FUNCTION_BLOCK ObserveSSC EXTENDS HardwareObservationBase
VAR_INPUT
END_VAR
VAR_OUTPUT
END_VAR
VAR
	m_ptrSSC: POINTER TO SmallSortingConveyor;
	m_ptrSSCWP1: POINTER TO xPPUProduct;
	m_ptrSSCWP2: POINTER TO xPPUProduct;
	
	m_rtWpAtRamp: R_TRIG;
END_VAR

METHOD FB_init : BOOL
VAR_INPUT
	bInitRetains : BOOL; // if TRUE, the retain variables are initialized (warm start / cold start)
	bInCopyCode : BOOL;  // if TRUE, the instance afterwards gets moved into the copy code (online change)
	
	i_ptrSSC: POINTER TO SmallSortingConveyor;
	i_ptrWP1: POINTER TO IProduct;
	i_ptrWP2: POINTER TO IProduct;
END_VAR
m_ptrSSC := i_ptrSSC;
IF NOT __QUERYPOINTER(i_ptrWP1^, m_ptrSSCWP1) THEN
	FB_init := FALSE;
END_IF
IF NOT __QUERYPOINTER(i_ptrWP2^, m_ptrSSCWP2) THEN
	FB_init := FALSE;
END_IF
END_METHOD

METHOD  ResetDefinition : BOOL
VAR_INPUT
END_VAR
;
END_METHOD

(* Update an instance of ProcessState with the part of the process that can be observed by this Hardware Interface. *)
METHOD UpdateProcessObservation : BOOL
VAR_IN_OUT
	io_processState: ProcessState;
END_VAR
m_rtWpAtRamp(CLK := m_ptrSSC^.WPAtRampEnd);

io_processState.UpdateState_Binary(EProcessVariables.SSC_WPAtStart, m_ptrSSC^.WPAtStart, TRUE);
io_processState.UpdateState_Binary(EProcessVariables.SSC_WPAtEnd, m_ptrSSC^.WPAtEnd, TRUE);
io_processState.UpdateState_Binary(EProcessVariables.SSC_WPLightAtMiddle, m_ptrSSC^.LightWPAtMid, TRUE);
io_processState.UpdateState_Binary(EProcessVariables.SSC_WPMetalAtMiddle, m_ptrSSC^.MetalWPAtMid, TRUE);
io_processState.UpdateState_Binary(EProcessVariables.SSC_WPAtRampEnd, m_ptrSSC^.WPAtRampEnd, TRUE);
io_processState.UpdateState_Binary(EProcessVariables.SSC_SwitchExtended, m_ptrSSC^.m_Switch.Extended, TRUE);
io_processState.UpdateState_Binary(EProcessVariables.SSC_SwitchRetracted, m_ptrSSC^.m_Switch.Retracted, TRUE);

IF m_rtWpAtRamp.Q THEN
	io_processState.UpdateState_NumericIncrement(EProcessVariables.SSC_RampWPCount, TRUE);
END_IF


io_processState.UpdateState_Defined(EProcessVariables.SSC_WPAtStart, TRUE);
io_processState.UpdateState_Defined(EProcessVariables.SSC_WPAtEnd, TRUE);
io_processState.UpdateState_Defined(EProcessVariables.SSC_WPLightAtMiddle, TRUE);
io_processState.UpdateState_Defined(EProcessVariables.SSC_WPMetalAtMiddle, TRUE);
io_processState.UpdateState_Defined(EProcessVariables.SSC_WPAtRampEnd, TRUE);
io_processState.UpdateState_Defined(EProcessVariables.SSC_SwitchExtended, TRUE);
io_processState.UpdateState_Defined(EProcessVariables.SSC_SwitchRetracted, TRUE);
// TODO - the following is technically not defined but how can we avoid that?
io_processState.UpdateState_Defined(EProcessVariables.SSC_RampWPCount, TRUE);


// update WP info (if there are sensors available), then update the process variables list

io_processState.UpdateState_Numeric(EProcessVariables.SSC_ProductType_1, UINT_TO_LREAL(m_ptrSSCWP1^.Material), TRUE);
io_processState.UpdateState_Numeric(EProcessVariables.SSC_ProductType_2, UINT_TO_LREAL(m_ptrSSCWP2^.Material), TRUE);

io_processState.UpdateState_Defined(EprocessVariables.SSC_ProductType_1, TRUE);
io_processState.UpdateState_Defined(EProcessVariables.SSC_ProductType_2, TRUE);
END_METHOD

END_FUNCTION_BLOCK

(* stored: Version 1.1.0.1, ProductVersion 3.1.4024.12
   POU ObserveSSC: Id {66efb86e-0f55-4957-be87-625d71a455b3}, SpecialFunc None
   Method FB_init: Id {b7cec3e1-cf3b-4b8f-99ec-0f0dfde818b5}
   Method ResetDefinition: Id {454d5de4-3775-456f-8448-2f51238c8a30}
   Method UpdateProcessObservation: Id {a96c4790-5b4e-41ac-814c-9aa10148e31c} *)
